# EPICS autosave request: iocBoot/generic_motors_ioc/dbSave/CS_Av_.req
%
% BURT Request File
%
% $(P)CS:Av:  Collimator (Monochromatic) slits, Vertical Aperture
%

file assy.req ASSY=$(P)CS:Av
$(P)CS:Av:Invert
file mtr1.req MTR1=$(P)CS:mz1
file mtr1.req MTR1=$(P)CS:mz2
file drv1.req DRV1=$(P)CS:ZT
file drv1.req DRV1=$(P)CS:ZB
file axs1.req AXS1=$(P)CS:ZC
file axs1.req AXS1=$(P)CS:ZS
